Fanuc KAREL source: DET_WINDOW.kl

PROGRAM T
%NOLOCKGROUP
VAR
 v0 : STRING[40]
 v1 : STRING[40]
 v2 : INTEGER
BEGIN
 DET_WINDOW(v0, v1, v2)
END T
